(* IEC 61131-3 sources: Easy_TwincatHMI/, 3 files *)

(* ---- example_struct_plc_code.st ---- *)
(*
    TwinCAT 3 PLC Example Code with STRUCT/DUT Auto-Import
    Demonstrates how to use HMI_STRUCT attribute for automatic struct import
*)

// ========================================
// STRUCT DEFINITIONS (DUT - Data Unit Types)
// ========================================

(*
    Analog Input Struct
    Used for temperature, pressure, flow sensors, etc.
*)
TYPE ST_AnalogInput :
STRUCT
    // Process value - will be imported as Process Value widget
    {attribute 'HMI_PV'}
    {attribute 'Unit' := '°C'}
    {attribute 'Decimals' := '2'}
    {attribute 'AlarmHighHigh' := '100'}
    {attribute 'AlarmHigh' := '90'}
    {attribute 'AlarmLow' := '5'}
    {attribute 'AlarmLowLow' := '2'}
    {attribute 'AlarmPriority' := '1'}
    Value : REAL;

    // Scaled value (0-100%)
    {attribute 'HMI_PV'}
    {attribute 'Unit' := '%'}
    {attribute 'Decimals' := '1'}
    Scaled : REAL;

    // Sensor error alarm
    {attribute 'HMI_ALARM'}
    {attribute 'AlarmText' := 'Sensor Kommunikationsfejl'}
    {attribute 'AlarmPriority' := '2'}
    Error : BOOL;

    // Calibration offset setpoint
    {attribute 'HMI_SP'}
    {attribute 'Unit' := 'Offset'}
    {attribute 'Min' := '-10'}
    {attribute 'Max' := '10'}
    {attribute 'Decimals' := '2'}
    {attribute 'Step' := '0.1'}
    CalibrationOffset : REAL;

    // Internal values - NOT imported (no HMI attribute)
    RawValue : INT;
    LastUpdateTime : TIME;
    SampleCount : UDINT;
END_STRUCT
END_TYPE

(*
    Motor Control Struct
    Complete motor control with setpoints and feedback
*)
TYPE ST_Motor :
STRUCT
    // Speed setpoint
    {attribute 'HMI_SP'}
    {attribute 'Unit' := 'RPM'}
    {attribute 'Min' := '0'}
    {attribute 'Max' := '3000'}
    {attribute 'Decimals' := '0'}
    {attribute 'Step' := '10'}
    SpeedSetpoint : REAL;

    // Actual speed
    {attribute 'HMI_PV'}
    {attribute 'Unit' := 'RPM'}
    {attribute 'Decimals' := '0'}
    {attribute 'AlarmHigh' := '3100'}
    ActualSpeed : REAL;

    // Current consumption
    {attribute 'HMI_PV'}
    {attribute 'Unit' := 'A'}
    {attribute 'Decimals' := '1'}
    {attribute 'AlarmHigh' := '15'}
    Current : REAL;

    // Run command switch
    {attribute 'HMI_SWITCH'}
    {attribute 'Pos0' := 'Stop'}
    {attribute 'Pos1' := 'Start'}
    {attribute 'Pos2' := 'Reset'}
    Command : INT;

    // Fault alarm
    {attribute 'HMI_ALARM'}
    {attribute 'AlarmText' := 'Motor Fejl'}
    {attribute 'AlarmPriority' := '1'}
    Fault : BOOL;

    // Overload alarm
    {attribute 'HMI_ALARM'}
    {attribute 'AlarmText' := 'Motor Overbelastet'}
    {attribute 'AlarmPriority' := '2'}
    Overload : BOOL;

    // Internal state - NOT imported
    InternalState : INT;
    RunningHours : TIME;
END_STRUCT
END_TYPE

(*
    PID Controller Struct
    Nested struct example
*)
TYPE ST_PIDParams :
STRUCT
    {attribute 'HMI_SP'}
    {attribute 'Min' := '0'}
    {attribute 'Max' := '100'}
    {attribute 'Decimals' := '2'}
    Kp : REAL;

    {attribute 'HMI_SP'}
    {attribute 'Min' := '0'}
    {attribute 'Max' := '10'}
    {attribute 'Decimals' := '3'}
    Ki : REAL;

    {attribute 'HMI_SP'}
    {attribute 'Min' := '0'}
    {attribute 'Max' := '10'}
    {attribute 'Decimals' := '3'}
    Kd : REAL;
END_STRUCT
END_TYPE

TYPE ST_TempController :
STRUCT
    // Temperature setpoint
    {attribute 'HMI_SP'}
    {attribute 'Unit' := '°C'}
    {attribute 'Min' := '0'}
    {attribute 'Max' := '100'}
    {attribute 'Decimals' := '1'}
    {attribute 'Step' := '0.5'}
    Setpoint : REAL;

    // Temperature process value
    {attribute 'HMI_PV'}
    {attribute 'Unit' := '°C'}
    {attribute 'Decimals' := '1'}
    {attribute 'AlarmHighHigh' := '98'}
    {attribute 'AlarmHigh' := '95'}
    ProcessValue : REAL;

    // Controller output
    {attribute 'HMI_PV'}
    {attribute 'Unit' := '%'}
    {attribute 'Decimals' := '1'}
    Output : REAL;

    // PID parameters (nested struct)
    // Note: PID members will also be imported if ST_PIDParams has HMI attributes
    PID : ST_PIDParams;

    // Control mode
    {attribute 'HMI_SWITCH'}
    {attribute 'Pos0' := 'Off'}
    {attribute 'Pos1' := 'Manual'}
    {attribute 'Pos2' := 'Automatic'}
    Mode : INT;
END_STRUCT
END_TYPE

(*
    Tank Level Monitoring
    Simple struct for level sensors
*)
TYPE ST_Tank :
STRUCT
    {attribute 'HMI_PV'}
    {attribute 'Unit' := '%'}
    {attribute 'Decimals' := '1'}
    {attribute 'AlarmHigh' := '90'}
    {attribute 'AlarmLow' := '10'}
    Level : REAL;

    {attribute 'HMI_PV'}
    {attribute 'Unit' := 'L'}
    {attribute 'Decimals' := '0'}
    Volume : REAL;

    {attribute 'HMI_ALARM'}
    {attribute 'AlarmText' := 'Tank Overfyldt'}
    {attribute 'AlarmPriority' := '1'}
    OverflowAlarm : BOOL;

    {attribute 'HMI_ALARM'}
    {attribute 'AlarmText' := 'Tank Næsten Tom'}
    {attribute 'AlarmPriority' := '3'}
    LowLevelWarning : BOOL;
END_STRUCT
END_TYPE

// ========================================
// GLOBAL VARIABLES WITH HMI_STRUCT MARKER
// ========================================

{attribute 'qualified_only'}
VAR_GLOBAL

    // ========================================
    // TEMPERATURE SENSORS
    // ========================================

    // Temperature sensor 1 - Auto-import entire struct
    {attribute 'HMI_STRUCT'}
    Temperature_Sensor_1 : ST_AnalogInput;

    // Temperature sensor 2
    {attribute 'HMI_STRUCT'}
    Temperature_Sensor_2 : ST_AnalogInput;

    // Pressure sensor
    {attribute 'HMI_STRUCT'}
    Pressure_Sensor_1 : ST_AnalogInput;

    // Flow sensor
    {attribute 'HMI_STRUCT'}
    Flow_Sensor_1 : ST_AnalogInput;

    // ========================================
    // MOTORS
    // ========================================

    // Main pump motor
    {attribute 'HMI_STRUCT'}
    Pump_Motor_1 : ST_Motor;

    // Backup pump motor
    {attribute 'HMI_STRUCT'}
    Pump_Motor_2 : ST_Motor;

    // Fan motor
    {attribute 'HMI_STRUCT'}
    Fan_Motor : ST_Motor;

    // ========================================
    // TEMPERATURE CONTROLLER
    // ========================================

    // Temperature controller (with nested PID params)
    {attribute 'HMI_STRUCT'}
    Temp_Controller_1 : ST_TempController;

    // ========================================
    // TANKS
    // ========================================

    // Storage tanks
    {attribute 'HMI_STRUCT'}
    Tank_1 : ST_Tank;

    {attribute 'HMI_STRUCT'}
    Tank_2 : ST_Tank;

    {attribute 'HMI_STRUCT'}
    Tank_3 : ST_Tank;

    // ========================================
    // ARRAY OF STRUCTS EXAMPLE
    // ========================================

    // Array of analog inputs
    {attribute 'HMI_STRUCT_ARRAY'}
    AnalogInputs : ARRAY[1..8] OF ST_AnalogInput;

    // ========================================
    // NON-HMI VARIABLES (not imported)
    // ========================================

    // These variables don't have HMI_STRUCT, so won't be auto-imported
    InternalCounter : UDINT;
    SystemState : INT;
    DebugFlags : WORD;

END_VAR

(*
    EXPECTED HMI IMPORT RESULT:

    When you click "Scan PLC" in the HMI application, it will find:

    GROUP: Temperature_Sensor_1 (ST_AnalogInput)
      ├─ Value              (Process Value, °C)
      ├─ Scaled             (Process Value, %)
      ├─ Error              (Alarm: Sensor Kommunikationsfejl)
      └─ CalibrationOffset  (Setpoint, Offset)

    GROUP: Temperature_Sensor_2 (ST_AnalogInput)
      ├─ Value              (Process Value, °C)
      ├─ Scaled             (Process Value, %)
      ├─ Error              (Alarm: Sensor Kommunikationsfejl)
      └─ CalibrationOffset  (Setpoint, Offset)

    GROUP: Pressure_Sensor_1 (ST_AnalogInput)
      ├─ Value              (Process Value, °C)
      ├─ Scaled             (Process Value, %)
      ├─ Error              (Alarm: Sensor Kommunikationsfejl)
      └─ CalibrationOffset  (Setpoint, Offset)

    GROUP: Pump_Motor_1 (ST_Motor)
      ├─ SpeedSetpoint      (Setpoint, RPM)
      ├─ ActualSpeed        (Process Value, RPM)
      ├─ Current            (Process Value, A)
      ├─ Command            (Switch: Stop/Start/Reset)
      ├─ Fault              (Alarm: Motor Fejl)
      └─ Overload           (Alarm: Motor Overbelastet)

    GROUP: Temp_Controller_1 (ST_TempController)
      ├─ Setpoint           (Setpoint, °C)
      ├─ ProcessValue       (Process Value, °C)
      ├─ Output             (Process Value, %)
      ├─ PID.Kp             (Setpoint)
      ├─ PID.Ki             (Setpoint)
      ├─ PID.Kd             (Setpoint)
      └─ Mode               (Switch: Off/Manual/Automatic)

    GROUP: Tank_1 (ST_Tank)
      ├─ Level              (Process Value, %)
      ├─ Volume             (Process Value, L)
      ├─ OverflowAlarm      (Alarm: Tank Overfyldt)
      └─ LowLevelWarning    (Alarm: Tank Næsten Tom)

    And similar groups for all other structs marked with {attribute 'HMI_STRUCT'}

    IMPORTANT NOTES:

    1. Only members with HMI attributes are imported:
       - HMI_SP, HMI_PV, HMI_SWITCH, HMI_ALARM
       - Members like RawValue, InternalState are skipped

    2. Full path is used for access:
       - Temperature_Sensor_1.Value
       - Pump_Motor_1.SpeedSetpoint
       - Temp_Controller_1.PID.Kp (nested)

    3. Config is automatically generated in config.json

    4. GUI widgets are automatically created and grouped

    5. All alarm limits, units, ranges are preserved from PLC
*)

(*
    USAGE INSTRUCTIONS:

    1. Copy these struct definitions to your TwinCAT project

    2. Copy the VAR_GLOBAL declarations

    3. Compile the TwinCAT project (F7)
       - This generates/updates the PLC.tmc file

    4. Set tmc_file path in HMI config.json:
       "tmc_file": "C:\\Path\\To\\Your\\Project\\PLC.tmc"

    5. Start the HMI application:
       py main.py

    6. Click "Forbind" to connect to PLC

    7. Click "Scan PLC" button
       - Application scans for symbols with HMI_STRUCT
       - Expands structs to members
       - Generates configuration
       - Creates GUI widgets

    8. Done! All struct members are now available in the HMI

    ADVANTAGES:

    ✅ Define struct once, use many times
    ✅ Consistent structure across multiple instances
    ✅ Easy to add new sensors/motors
    ✅ No manual HMI configuration needed
    ✅ Type-safe (PLC compiler checks)
    ✅ Automatic GUI grouping
    ✅ All metadata from PLC attributes

    BEST PRACTICES:

    1. Use descriptive struct names (ST_AnalogInput, ST_Motor)
    2. Add HMI attributes to relevant members only
    3. Use consistent naming (Setpoint, ProcessValue, Error)
    4. Group related functionality in structs
    5. Document struct purpose in comments
    6. Test with one struct before creating many
*)

(* ---- motor_fb_example.st ---- *)
(*
================================================================================
    MOTOR FUNCTION BLOCK WITH HMI INTEGRATION

    Description: Complete motor control function block with:
    - Start/Stop control with safety interlocks
    - Speed control with ramping
    - Start frequency monitoring and protection
    - Feedback monitoring with alarms
    - Full HMI integration using structured attributes

    Author: TwinCAT HMI Example
    Date: 2025-01-28
================================================================================
*)

// ============================================================================
// TYPE DEFINITIONS
// ============================================================================

TYPE ST_MotorCommands :
STRUCT
    {attribute 'HMI_CMD'}
    {attribute 'CmdText' := 'Start Motor'}
    Start : BOOL := FALSE;          // Start command from HMI

    {attribute 'HMI_CMD'}
    {attribute 'CmdText' := 'Stop Motor'}
    Stop : BOOL := FALSE;           // Stop command from HMI

    {attribute 'HMI_CMD'}
    {attribute 'CmdText' := 'Reset Alarms'}
    Reset : BOOL := FALSE;          // Reset all alarms and errors

    {attribute 'HMI_SP'}
    {attribute 'Unit' := '%'}
    {attribute 'Min' := '0'}
    {attribute 'Max' := '100'}
    {attribute 'Decimals' := '1'}
    {attribute 'Step' := '1'}
    SpeedSetpoint : REAL := 0.0;    // Speed setpoint 0-100%
END_STRUCT
END_TYPE

TYPE ST_MotorSettings :
STRUCT
    {attribute 'HMI_SP'}
    {attribute 'Unit' := 'Starts/min'}
    {attribute 'Min' := '1'}
    {attribute 'Max' := '10'}
    {attribute 'Decimals' := '0'}
    {attribute 'Step' := '1'}
    MaxStartsPerMinute : INT := 6;          // Max allowed starts per minute

    {attribute 'HMI_SP'}
    {attribute 'Unit' := 's'}
    {attribute 'Min' := '10'}
    {attribute 'Max' := '600'}
    {attribute 'Decimals' := '0'}
    {attribute 'Step' := '10'}
    MaxTimeAtMaxStarts : TIME := T#60S;     // Max time in alarm before shutdown

    {attribute 'HMI_SP'}
    {attribute 'Unit' := '%'}
    {attribute 'Min' := '0'}
    {attribute 'Max' := '100'}
    {attribute 'Decimals' := '1'}
    {attribute 'Step' := '5'}
    MaxStartSpeed : REAL := 50.0;           // Max speed during start sequence

    {attribute 'HMI_SP'}
    {attribute 'Unit' := 'ms'}
    {attribute 'Min' := '10'}
    {attribute 'Max' := '1000'}
    {attribute 'Decimals' := '0'}
    {attribute 'Step' := '10'}
    RampTimePerPercent : TIME := T#50MS;    // Time per 1% speed change

    {attribute 'HMI_SP'}
    {attribute 'Unit' := 's'}
    {attribute 'Min' := '1'}
    {attribute 'Max' := '30'}
    {attribute 'Decimals' := '1'}
    {attribute 'Step' := '0.5'}
    FeedbackTimeout : TIME := T#5S;         // Time to reach target speed

    {attribute 'HMI_SP'}
    {attribute 'Unit' := '%'}
    {attribute 'Min' := '1'}
    {attribute 'Max' := '20'}
    {attribute 'Decimals' := '1'}
    {attribute 'Step' := '0.5'}
    FeedbackTolerance : REAL := 5.0;        // Acceptable speed deviation
END_STRUCT
END_TYPE

TYPE ST_MotorFeedback :
STRUCT
    {attribute 'HMI_PV'}
    Running : BOOL := FALSE;                // Motor is running

    {attribute 'HMI_PV'}
    {attribute 'Unit' := '%'}
    {attribute 'Decimals' := '1'}
    ActualSpeed : REAL := 0.0;              // Actual motor speed 0-100%

    {attribute 'HMI_PV'}
    ThermalRelay : BOOL := FALSE;           // Thermal relay status (TRUE = OK)

    {attribute 'HMI_PV'}
    Thermistor : BOOL := FALSE;             // Thermistor status (TRUE = OK)

    {attribute 'HMI_PV'}
    VFD_Ready : BOOL := FALSE;              // VFD ready status

    {attribute 'HMI_PV'}
    VFD_Fault : BOOL := FALSE;              // VFD fault status

    {attribute 'HMI_PV'}
    {attribute 'Unit' := 'Starts'}
    {attribute 'Decimals' := '0'}
    StartCountLastMinute : INT := 0;        // Start count in last minute
END_STRUCT
END_TYPE

TYPE ST_MotorAlarms :
STRUCT
    {attribute 'HMI_ALARM'}
    {attribute 'AlarmText' := 'For mange opstart per minut'}
    {attribute 'AlarmPriority' := '2'}
    {attribute 'AlarmActive' := TRUE}
    {attribute 'WarningActive' := FALSE}
    TooManyStarts : BOOL := FALSE;          // Too many starts alarm

    {attribute 'HMI_ALARM'}
    {attribute 'AlarmText' := 'Motor stoppet - for mange opstart'}
    {attribute 'AlarmPriority' := '1'}
    {attribute 'AlarmActive' := TRUE}
    {attribute 'WarningActive' := FALSE}
    StartProtectionShutdown : BOOL := FALSE; // Protection shutdown

    {attribute 'HMI_ALARM'}
    {attribute 'AlarmText' := 'Hastighedsfeedback fejl'}
    {attribute 'AlarmPriority' := '2'}
    {attribute 'AlarmActive' := TRUE}
    {attribute 'WarningActive' := FALSE}
    SpeedFeedbackFault : BOOL := FALSE;     // Speed not reached in time

    {attribute 'HMI_ALARM'}
    {attribute 'AlarmText' := 'Termorelæ udløst'}
    {attribute 'AlarmPriority' := '1'}
    {attribute 'AlarmActive' := TRUE}
    {attribute 'WarningActive' := FALSE}
    ThermalRelayTripped : BOOL := FALSE;    // Thermal protection

    {attribute 'HMI_ALARM'}
    {attribute 'AlarmText' := 'Termistor fejl'}
    {attribute 'AlarmPriority' := '1'}
    {attribute 'AlarmActive' := TRUE}
    {attribute 'WarningActive' := FALSE}
    ThermistorFault : BOOL := FALSE;        // Motor overtemperature

    {attribute 'HMI_ALARM'}
    {attribute 'AlarmText' := 'VFD fejl'}
    {attribute 'AlarmPriority' := '1'}
    {attribute 'AlarmActive' := TRUE}
    {attribute 'WarningActive' := FALSE}
    VFD_Fault : BOOL := FALSE;              // Variable frequency drive fault
END_STRUCT
END_TYPE

// ============================================================================
// FUNCTION BLOCK
// ============================================================================

FUNCTION_BLOCK FB_Motor
VAR_INPUT
    // Physical inputs from motor and VFD
    I_ThermalRelay      : BOOL;     // Thermal relay contact (TRUE = OK)
    I_Thermistor        : BOOL;     // Thermistor input (TRUE = OK)
    I_VFD_Ready         : BOOL;     // VFD ready signal
    I_VFD_Fault         : BOOL;     // VFD fault signal
    I_SpeedFeedback     : REAL;     // Speed feedback from VFD (0-100%)
    I_Enable            : BOOL;     // External enable signal
END_VAR

VAR_OUTPUT
    // Physical outputs to motor and VFD
    Q_Start             : BOOL;     // Start output to VFD
    Q_SpeedReference    : REAL;     // Speed reference to VFD (0-100%)
    Q_Fault             : BOOL;     // General fault output
END_VAR

VAR_IN_OUT
    // HMI interface structures
    Commands    : ST_MotorCommands;
    Settings    : ST_MotorSettings;
    Feedback    : ST_MotorFeedback;
    Alarms      : ST_MotorAlarms;
END_VAR

VAR
    // Internal state machine
    State               : INT := 0;

    // Ramping control
    CurrentSpeed        : REAL := 0.0;
    TargetSpeed         : REAL := 0.0;
    RampTimer           : TON;

    // Start frequency monitoring
    StartTimeStamps     : ARRAY[1..20] OF TIME;
    StartIndex          : INT := 1;
    TooManyStartsTimer  : TON;

    // Feedback monitoring
    FeedbackTimer       : TON;
    SpeedReached        : BOOL := FALSE;

    // Edge detection
    StartCmd_R_TRIG     : R_TRIG;
    StopCmd_R_TRIG      : R_TRIG;
    ResetCmd_R_TRIG     : R_TRIG;

    // Timers
    CurrentTime         : TIME;
END_VAR

VAR CONSTANT
    STATE_STOPPED       : INT := 0;
    STATE_STARTING      : INT := 1;
    STATE_RUNNING       : INT := 2;
    STATE_STOPPING      : INT := 3;
    STATE_FAULT         : INT := 4;
END_VAR

(*
================================================================================
    Main Program Logic
================================================================================
*)

// Get current system time
CurrentTime := TIME();

// Edge detection for commands
StartCmd_R_TRIG(CLK := Commands.Start);
StopCmd_R_TRIG(CLK := Commands.Stop);
ResetCmd_R_TRIG(CLK := Commands.Reset);

// Reset command handling
IF ResetCmd_R_TRIG.Q THEN
    // Reset all alarms
    Alarms.TooManyStarts := FALSE;
    Alarms.StartProtectionShutdown := FALSE;
    Alarms.SpeedFeedbackFault := FALSE;
    Alarms.ThermalRelayTripped := FALSE;
    Alarms.ThermistorFault := FALSE;
    Alarms.VFD_Fault := FALSE;

    // Reset to stopped state if not in critical fault
    IF State = STATE_FAULT THEN
        State := STATE_STOPPED;
    END_IF;

    // Reset command (self-clearing)
    Commands.Reset := FALSE;
END_IF;

// Update feedback from physical inputs
Feedback.ThermalRelay := I_ThermalRelay;
Feedback.Thermistor := I_Thermistor;
Feedback.VFD_Ready := I_VFD_Ready;
Feedback.VFD_Fault := I_VFD_Fault;
Feedback.ActualSpeed := I_SpeedFeedback;

// Check for hardware faults
IF NOT I_ThermalRelay THEN
    Alarms.ThermalRelayTripped := TRUE;
    State := STATE_FAULT;
END_IF;

IF NOT I_Thermistor THEN
    Alarms.ThermistorFault := TRUE;
    State := STATE_FAULT;
END_IF;

IF I_VFD_Fault THEN
    Alarms.VFD_Fault := TRUE;
    State := STATE_FAULT;
END_IF;

// Start frequency protection monitoring
MonitorStartFrequency();

// State machine
CASE State OF

    STATE_STOPPED:
        // Stopped state
        CurrentSpeed := 0.0;
        TargetSpeed := 0.0;
        Q_Start := FALSE;
        Q_SpeedReference := 0.0;
        Feedback.Running := FALSE;
        SpeedReached := FALSE;

        // Check if start is allowed
        IF StartCmd_R_TRIG.Q AND I_Enable AND I_VFD_Ready AND NOT Alarms.StartProtectionShutdown THEN
            // Log start time
            LogStartTime();

            // Limit target speed during start sequence
            IF Commands.SpeedSetpoint > Settings.MaxStartSpeed THEN
                TargetSpeed := Settings.MaxStartSpeed;
            ELSE
                TargetSpeed := Commands.SpeedSetpoint;
            END_IF;

            State := STATE_STARTING;
        END_IF;

        // Clear start command
        Commands.Start := FALSE;

    STATE_STARTING:
        // Starting state
        Q_Start := TRUE;

        // Ramp up speed
        IF CurrentSpeed < TargetSpeed THEN
            RampSpeed(TRUE);
        ELSIF CurrentSpeed > TargetSpeed THEN
            RampSpeed(FALSE);
        ELSE
            // Speed reached
            State := STATE_RUNNING;
            SpeedReached := FALSE;
        END_IF;

        // Monitor speed feedback
        MonitorSpeedFeedback();

        // Check for stop command
        IF StopCmd_R_TRIG.Q OR NOT I_Enable THEN
            State := STATE_STOPPING;
        END_IF;

        // Clear stop command
        Commands.Stop := FALSE;

    STATE_RUNNING:
        // Running state
        Q_Start := TRUE;
        Feedback.Running := TRUE;

        // Update target speed from setpoint
        TargetSpeed := Commands.SpeedSetpoint;

        // Ramp to target speed
        IF CurrentSpeed < TargetSpeed THEN
            RampSpeed(TRUE);
        ELSIF CurrentSpeed > TargetSpeed THEN
            RampSpeed(FALSE);
        END_IF;

        // Monitor speed feedback
        MonitorSpeedFeedback();

        // Check for stop command
        IF StopCmd_R_TRIG.Q OR NOT I_Enable THEN
            State := STATE_STOPPING;
        END_IF;

        // Clear stop command
        Commands.Stop := FALSE;

    STATE_STOPPING:
        // Stopping state
        Q_Start := FALSE;
        TargetSpeed := 0.0;

        // Ramp down speed
        IF CurrentSpeed > 0.0 THEN
            RampSpeed(FALSE);
        ELSE
            // Fully stopped
            State := STATE_STOPPED;
        END_IF;

    STATE_FAULT:
        // Fault state - emergency stop
        Q_Start := FALSE;
        CurrentSpeed := 0.0;
        TargetSpeed := 0.0;
        Q_SpeedReference := 0.0;
        Feedback.Running := FALSE;
        Q_Fault := TRUE;

        // Can only exit fault state with reset command
        // Reset is handled above
END_CASE;

// Always output current speed reference
Q_SpeedReference := CurrentSpeed;

// Clear fault output if no active critical alarms
IF NOT (Alarms.ThermalRelayTripped OR Alarms.ThermistorFault OR Alarms.VFD_Fault OR Alarms.StartProtectionShutdown) THEN
    Q_Fault := FALSE;
END_IF;

// ============================================================================
// INTERNAL METHODS
// ============================================================================

(*
    RampSpeed - Ramps speed up or down based on ramp time setting
*)
METHOD PRIVATE RampSpeed
VAR_INPUT
    RampUp : BOOL;      // TRUE = ramp up, FALSE = ramp down
END_VAR

    // Start/restart ramp timer
    RampTimer(IN := TRUE, PT := Settings.RampTimePerPercent);

    IF RampTimer.Q THEN
        // Time to increment/decrement speed
        IF RampUp THEN
            CurrentSpeed := CurrentSpeed + 1.0;
            IF CurrentSpeed > TargetSpeed THEN
                CurrentSpeed := TargetSpeed;
            END_IF;
            IF CurrentSpeed > 100.0 THEN
                CurrentSpeed := 100.0;
            END_IF;
        ELSE
            CurrentSpeed := CurrentSpeed - 1.0;
            IF CurrentSpeed < TargetSpeed THEN
                CurrentSpeed := TargetSpeed;
            END_IF;
            IF CurrentSpeed < 0.0 THEN
                CurrentSpeed := 0.0;
            END_IF;
        END_IF;

        // Reset timer for next step
        RampTimer(IN := FALSE);
    END_IF;
END_METHOD

(*
    MonitorSpeedFeedback - Monitors if actual speed reaches target
*)
METHOD PRIVATE MonitorSpeedFeedback

VAR
    SpeedError : REAL;
END_VAR

    SpeedError := ABS(TargetSpeed - I_SpeedFeedback);

    // Check if speed is within tolerance
    IF SpeedError <= Settings.FeedbackTolerance THEN
        SpeedReached := TRUE;
        FeedbackTimer(IN := FALSE);
        Alarms.SpeedFeedbackFault := FALSE;
    ELSE
        SpeedReached := FALSE;

        // Start timeout timer if not already reached
        FeedbackTimer(IN := TRUE, PT := Settings.FeedbackTimeout);

        // Check for timeout
        IF FeedbackTimer.Q THEN
            Alarms.SpeedFeedbackFault := TRUE;
        END_IF;
    END_IF;
END_METHOD

(*
    LogStartTime - Records timestamp of motor start
*)
METHOD PRIVATE LogStartTime

    // Store current time in circular buffer
    StartTimeStamps[StartIndex] := CurrentTime;
    StartIndex := StartIndex + 1;

    // Wrap around buffer
    IF StartIndex > 20 THEN
        StartIndex := 1;
    END_IF;
END_METHOD

(*
    MonitorStartFrequency - Monitors number of starts per minute
*)
METHOD PRIVATE MonitorStartFrequency

VAR
    i : INT;
    StartCount : INT := 0;
    TimeWindow : TIME := T#60S;
END_VAR

    // Count starts within last minute
    FOR i := 1 TO 20 DO
        IF (CurrentTime - StartTimeStamps[i]) <= TimeWindow AND StartTimeStamps[i] > T#0S THEN
            StartCount := StartCount + 1;
        END_IF;
    END_FOR;

    // Update feedback
    Feedback.StartCountLastMinute := StartCount;

    // Check if too many starts
    IF StartCount >= Settings.MaxStartsPerMinute THEN
        Alarms.TooManyStarts := TRUE;

        // Start protection timer
        TooManyStartsTimer(IN := TRUE, PT := Settings.MaxTimeAtMaxStarts);

        // Check if timer expired - trigger shutdown
        IF TooManyStartsTimer.Q THEN
            Alarms.StartProtectionShutdown := TRUE;
            State := STATE_FAULT;
            TooManyStartsTimer(IN := FALSE);
        END_IF;
    ELSE
        Alarms.TooManyStarts := FALSE;
        TooManyStartsTimer(IN := FALSE);
    END_IF;
END_METHOD

END_FUNCTION_BLOCK

// ============================================================================
// USAGE EXAMPLE - Global Variable Declaration
// ============================================================================

(*
{attribute 'qualified_only'}
VAR_GLOBAL
    // Motor instance with all structures
    Motor1 : FB_Motor;

    // Motor command interface
    {attribute 'HMI_GROUP'}
    Motor1_Commands : ST_MotorCommands;

    // Motor settings
    {attribute 'HMI_GROUP'}
    Motor1_Settings : ST_MotorSettings;

    // Motor feedback
    {attribute 'HMI_GROUP'}
    Motor1_Feedback : ST_MotorFeedback;

    // Motor alarms
    {attribute 'HMI_GROUP'}
    Motor1_Alarms : ST_MotorAlarms;
END_VAR

// ============================================================================
// USAGE EXAMPLE - Main Program
// ============================================================================

PROGRAM MAIN
VAR
    // Physical I/O mappings (example)
    DI_Motor1_ThermalRelay  AT %I* : BOOL;
    DI_Motor1_Thermistor    AT %I* : BOOL;
    DI_Motor1_VFD_Ready     AT %I* : BOOL;
    DI_Motor1_VFD_Fault     AT %I* : BOOL;
    AI_Motor1_SpeedFB       AT %I* : REAL;

    DO_Motor1_Start         AT %Q* : BOOL;
    AO_Motor1_SpeedRef      AT %Q* : REAL;
    DO_Motor1_Fault         AT %Q* : BOOL;

    EnableMotor1            : BOOL := TRUE;
END_VAR

// Call motor function block
Motor1(
    I_ThermalRelay      := DI_Motor1_ThermalRelay,
    I_Thermistor        := DI_Motor1_Thermistor,
    I_VFD_Ready         := DI_Motor1_VFD_Ready,
    I_VFD_Fault         := DI_Motor1_VFD_Fault,
    I_SpeedFeedback     := AI_Motor1_SpeedFB,
    I_Enable            := EnableMotor1,
    Q_Start             => DO_Motor1_Start,
    Q_SpeedReference    => AO_Motor1_SpeedRef,
    Q_Fault             => DO_Motor1_Fault,
    Commands            := Motor1_Commands,
    Settings            := Motor1_Settings,
    Feedback            := Motor1_Feedback,
    Alarms              := Motor1_Alarms
);

END_PROGRAM
*)

(* ---- example_plc_code.st ---- *)
(*
    TwinCAT 3 PLC Example Code
    Example global variables with HMI attributes for alarm system
*)

{attribute 'qualified_only'}
VAR_GLOBAL

    // ========================================
    // SETPOINTS (HMI_SP)
    // ========================================

    // Temperature setpoint with alarms
    {attribute 'HMI_SP'}
    {attribute 'Unit' := '°C'}
    {attribute 'Min' := '0'}
    {attribute 'Max' := '100'}
    {attribute 'Decimals' := '1'}
    {attribute 'Step' := '0.5'}
    {attribute 'AlarmHighHigh' := '95'}      // Critical high alarm at 95°C
    {attribute 'AlarmHigh' := '85'}           // High alarm at 85°C
    {attribute 'AlarmLow' := '10'}            // Low alarm at 10°C
    {attribute 'AlarmLowLow' := '5'}          // Critical low alarm at 5°C
    {attribute 'AlarmPriority' := '1'}        // Priority 1 = Critical
    TemperaturSetpunkt : REAL := 25.0;

    // Pressure setpoint
    {attribute 'HMI_SP'}
    {attribute 'Unit' := 'bar'}
    {attribute 'Min' := '0'}
    {attribute 'Max' := '10'}
    {attribute 'Decimals' := '2'}
    {attribute 'AlarmHigh' := '9.5'}
    TrykSetpunkt : REAL := 5.0;

    // Flow setpoint
    {attribute 'HMI_SP'}
    {attribute 'Unit' := 'L/min'}
    {attribute 'Min' := '0'}
    {attribute 'Max' := '200'}
    {attribute 'Decimals' := '1'}
    FlowSetpunkt : REAL := 100.0;

    // ========================================
    // PROCESS VALUES (HMI_PV)
    // ========================================

    // Temperature process value with alarms
    {attribute 'HMI_PV'}
    {attribute 'Unit' := '°C'}
    {attribute 'Decimals' := '2'}
    {attribute 'AlarmHighHigh' := '98'}       // Critical high at 98°C
    {attribute 'AlarmHigh' := '90'}           // Warning high at 90°C
    {attribute 'AlarmLow' := '5'}             // Warning low at 5°C
    {attribute 'AlarmLowLow' := '2'}          // Critical low at 2°C
    {attribute 'AlarmPriority' := '1'}        // Critical priority
    Temperatur_1 : REAL := 23.5;

    // Second temperature sensor
    {attribute 'HMI_PV'}
    {attribute 'Unit' := '°C'}
    {attribute 'Decimals' := '2'}
    {attribute 'AlarmHighHigh' := '95'}
    {attribute 'AlarmHigh' := '85'}
    Temperatur_2 : REAL := 24.0;

    // Pressure with high alarm only
    {attribute 'HMI_PV'}
    {attribute 'Unit' := 'bar'}
    {attribute 'Decimals' := '2'}
    {attribute 'AlarmHigh' := '9.5'}
    {attribute 'AlarmPriority' := '2'}        // High priority
    Tryk_1 : REAL := 5.0;

    // Flow measurement
    {attribute 'HMI_PV'}
    {attribute 'Unit' := 'L/min'}
    {attribute 'Decimals' := '1'}
    {attribute 'AlarmHigh' := '180'}
    {attribute 'AlarmLow' := '20'}
    Flow_1 : REAL := 100.0;

    // Level measurement (no alarms)
    {attribute 'HMI_PV'}
    {attribute 'Unit' := '%'}
    {attribute 'Decimals' := '1'}
    Niveau_1 : REAL := 50.0;

    // ========================================
    // SWITCHES (HMI_SWITCH)
    // ========================================

    // Operating mode selector
    {attribute 'HMI_SWITCH'}
    {attribute 'Pos0' := 'Stop'}
    {attribute 'Pos1' := 'Auto'}
    {attribute 'Pos2' := 'Manuel'}
    DriftMode : INT := 1;

    // Pump selector
    {attribute 'HMI_SWITCH'}
    {attribute 'Pos0' := 'Off'}
    {attribute 'Pos1' := 'Pumpe 1'}
    {attribute 'Pos2' := 'Pumpe 2'}
    {attribute 'Pos3' := 'Begge'}
    PumpeValg : INT := 0;

    // Priority selector
    {attribute 'HMI_SWITCH'}
    {attribute 'Pos0' := 'Normal'}
    {attribute 'Pos1' := 'Høj'}
    {attribute 'Pos2' := 'Kritisk'}
    Prioritet : INT := 0;

    // ========================================
    // DIGITAL ALARMS (HMI_ALARM)
    // ========================================

    // Motor fault alarm
    {attribute 'HMI_ALARM'}
    {attribute 'AlarmText' := 'Motor 1 Fejl'}
    {attribute 'AlarmPriority' := '1'}        // Critical
    Motor1Fejl : BOOL := FALSE;

    // Emergency stop
    {attribute 'HMI_ALARM'}
    {attribute 'AlarmText' := 'Nødstop Aktiveret'}
    {attribute 'AlarmPriority' := '1'}        // Critical
    NodStop : BOOL := FALSE;

    // Low oil pressure
    {attribute 'HMI_ALARM'}
    {attribute 'AlarmText' := 'Lavt Olietryk'}
    {attribute 'AlarmPriority' := '2'}        // High
    LavtOlieTryk : BOOL := FALSE;

    // Filter warning
    {attribute 'HMI_ALARM'}
    {attribute 'AlarmText' := 'Filter Skal Skiftes'}
    {attribute 'AlarmPriority' := '3'}        // Medium
    FilterAdvarsel : BOOL := FALSE;

    // Maintenance reminder
    {attribute 'HMI_ALARM'}
    {attribute 'AlarmText' := 'Vedligehold Nødvendigt'}
    {attribute 'AlarmPriority' := '4'}        // Low
    VedligeholdPaamindelse : BOOL := FALSE;

    // ========================================
    // STATUS FLAGS (No HMI attributes)
    // ========================================

    SystemRunning : BOOL := FALSE;
    ErrorCount : INT := 0;
    LastUpdateTime : TIME := T#0S;

END_VAR

(*
    USAGE NOTES:

    1. Copy this variable declaration to your TwinCAT project
    2. Compile the project
    3. Run the Python HMI application
    4. The HMI will automatically discover all variables with HMI_ attributes

    ATTRIBUTE REFERENCE:

    HMI_SP          - Setpoint (writable from HMI)
    HMI_PV          - Process Value (read-only)
    HMI_SWITCH      - Switch/Selector (writable)
    HMI_ALARM       - Digital alarm (BOOL)

    Unit            - Display unit
    Min/Max         - Valid range for setpoints
    Decimals        - Number of decimal places
    Step            - Increment step for spinbox

    AlarmHighHigh   - Critical high alarm limit
    AlarmHigh       - Warning high alarm limit
    AlarmLow        - Warning low alarm limit
    AlarmLowLow     - Critical low alarm limit
    AlarmPriority   - 1=Critical, 2=High, 3=Medium, 4=Low
    AlarmText       - Text for digital alarms

    Pos0, Pos1, etc - Switch position labels

    ALARM BEHAVIOR:

    - Alarms trigger when value crosses limit
    - Alarms clear with 2% hysteresis (configurable)
    - HighHigh and LowLow are critical (Priority 1)
    - High and Low are warnings (Priority 2)
    - Digital alarms trigger when BOOL = TRUE

    EXAMPLE TEST SEQUENCE:

    1. Set Temperatur_1 := 92.0  -> High alarm
    2. Set Temperatur_1 := 99.0  -> HighHigh (critical) alarm
    3. Set Motor1Fejl := TRUE    -> Critical digital alarm
    4. Acknowledge alarms in HMI
    5. Reset values to clear alarms
*)
